Fanuc KAREL source: kc00059.KL

-- PROVISIONAL review KL for V940-1; original PC SHA256 4700e0e1db01ca25f9ad0e915f8ed8d6edf0cc28b6c212d62d25606528bbd317
-- Incomplete behavior may be omitted. Consult companion uncertainty JSON. Do not deploy.
PROGRAM KC00059
%NOLOCKGROUP
BEGIN
  -- V9_ZERO_TABLE_METADATA_HINT layout=0002_ascii; no indexed target words; source/name/runtime held
  -- UNRESOLVED_PC offsets 5-25; opcodes 27,27,9D,27,9D,22,AA,23
  -- UNRESOLVED_PC offsets 30-34; opcodes 7F
END KC00059
